FUNCTION_BLOCK SS5b_Ejector (* Basic FB with empty ECC *)
  (* Standard: 61499-2 *)
  (* Version 1.0, 2024-10-03, DEVIASH *)
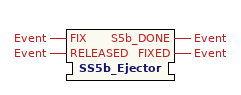
  EVENT_INPUT
    FIX;
    RELEASED;
  END_EVENT
  EVENT_OUTPUT
    S5b_DONE;
    FIXED;
  END_EVENT
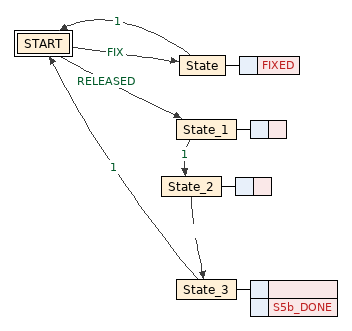
  EC_STATES
    START; (* Initial State *)
    State : -> FIXED;
    State_1;
    State_2;
    State_3 : -> S5b_DONE;
  END_STATES
  EC_TRANSITIONS
    START TO State := FIX;
    State TO START := 1;
    START TO State_1 := RELEASED;
    State_1 TO State_2 := 1;
    State_2 TO State_3 := ;
    State_3 TO START := 1;
  END_TRANSITIONS
END_FUNCTION_BLOCK
